# EPICS autosave request: iocBoot/iocGalilTest/GalilTest_DMC01Positions.req
$(P)A.DVAL
$(P)B.DVAL
$(P)C.DVAL
$(P)D.DVAL
$(P)E.DVAL
$(P)F.DVAL
$(P)G.DVAL
$(P)H.DVAL
